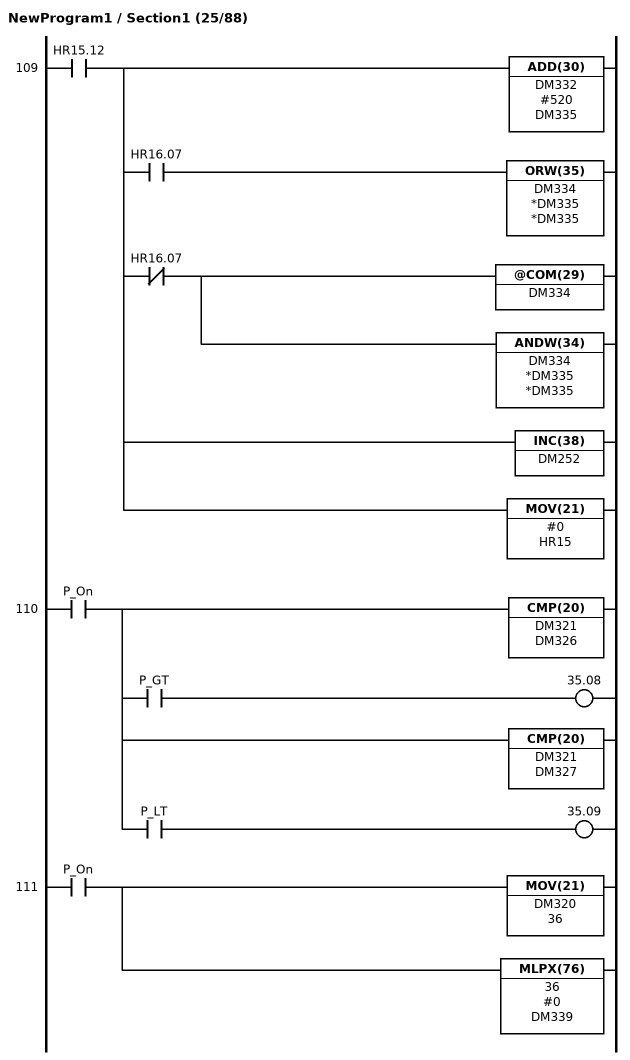
; [picture p24: NewProgram1 / Section1, rungs 109-111]
; rung 109
LD HR15.12
OUT TR0
ADD(30) DM332 #520 DM335
AND HR16.07
ORW(35) DM334 *DM335 *DM335
LD TR0
ANDNOT HR16.07
@COM(29) DM334
ANDW(34) DM334 *DM335 *DM335
LD TR0
INC(38) DM252
MOV(21) #0 HR15
; rung 110
LD P_On
OUT TR0
CMP(20) DM321 DM326
AND P_GT
OUT 35.08
LD TR0
CMP(20) DM321 DM327
AND P_LT
OUT 35.09
; rung 111
LD P_On
MOV(21) DM320 36
MLPX(76) 36 #0 DM339

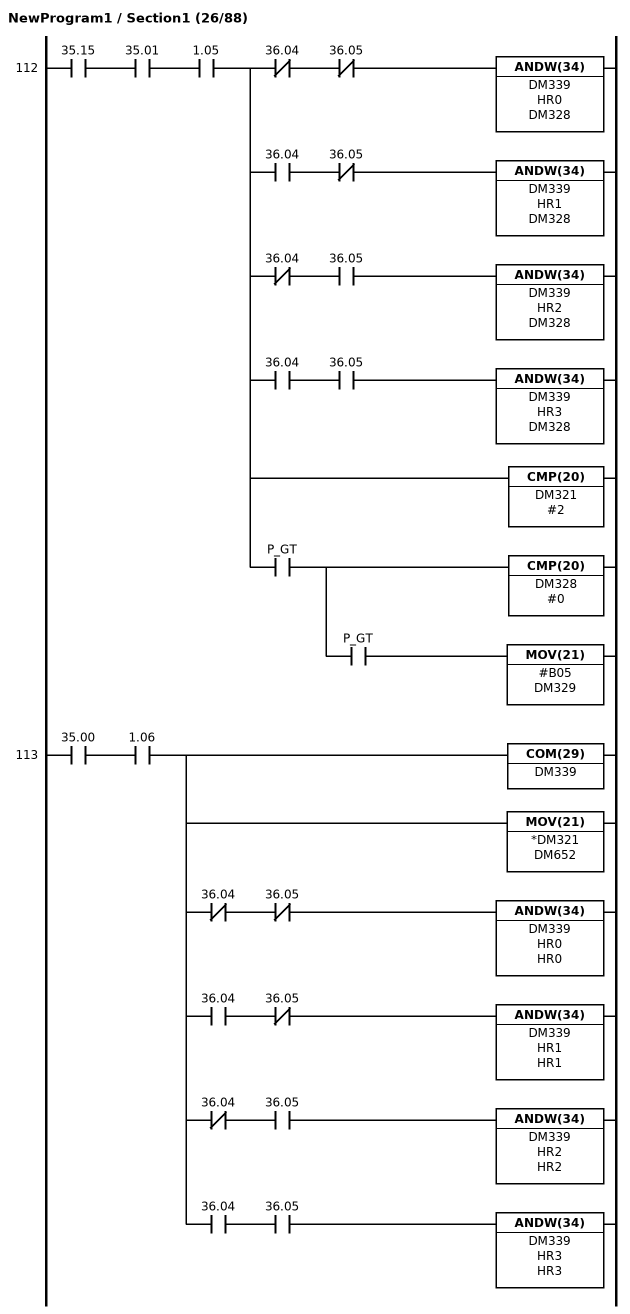
; rung 112
LD 35.15
AND 35.01
AND 1.05
OUT TR0
ANDNOT 36.04
ANDNOT 36.05
ANDW(34) DM339 HR0 DM328
LD TR0
AND 36.04
ANDNOT 36.05
ANDW(34) DM339 HR1 DM328
LD TR0
ANDNOT 36.04
AND 36.05
ANDW(34) DM339 HR2 DM328
LD TR0
AND 36.04
AND 36.05
ANDW(34) DM339 HR3 DM328
LD TR0
CMP(20) DM321 #2
AND P_GT
CMP(20) DM328 #0
AND P_GT
MOV(21) #B05 DM329
; rung 113
LD 35.00
AND 1.06
OUT TR0
COM(29) DM339
MOV(21) *DM321 DM652
ANDNOT 36.04
ANDNOT 36.05
ANDW(34) DM339 HR0 HR0
LD TR0
AND 36.04
ANDNOT 36.05
ANDW(34) DM339 HR1 HR1
LD TR0
ANDNOT 36.04
AND 36.05
ANDW(34) DM339 HR2 HR2
LD TR0
AND 36.04
AND 36.05
ANDW(34) DM339 HR3 HR3

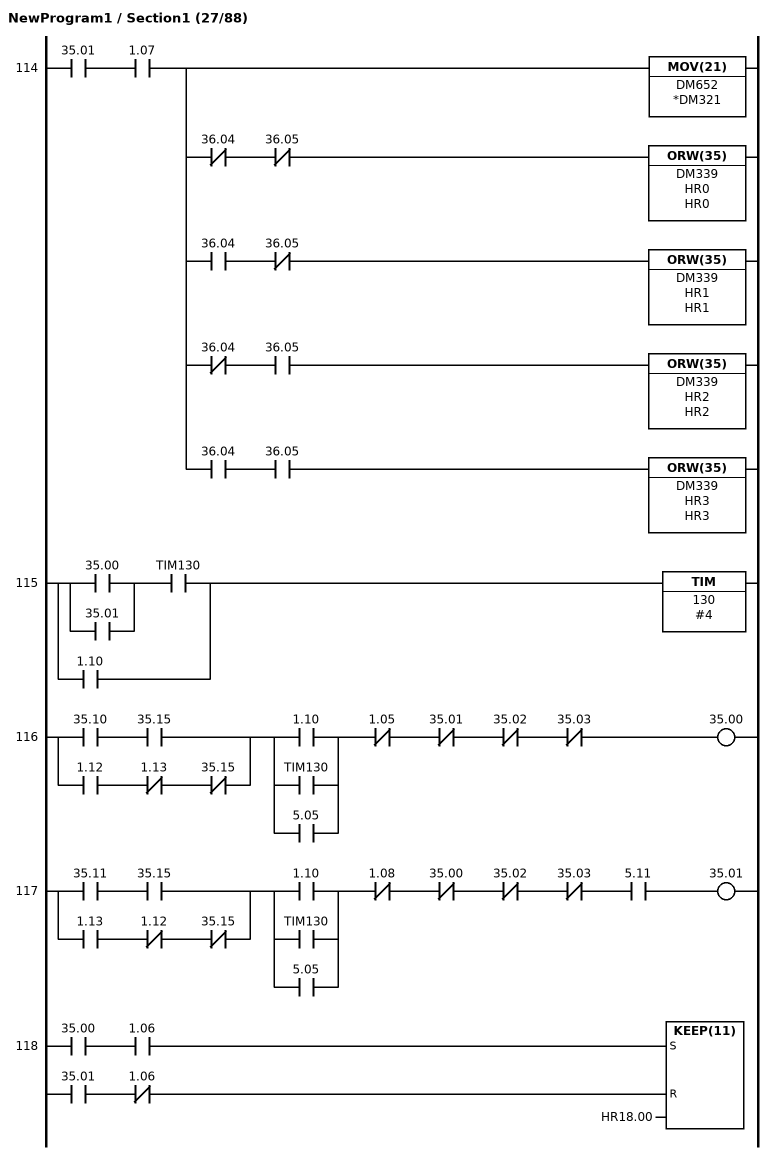
; rung 114
LD 35.01
AND 1.07
OUT TR0
MOV(21) DM652 *DM321
ANDNOT 36.04
ANDNOT 36.05
ORW(35) DM339 HR0 HR0
LD TR0
AND 36.04
ANDNOT 36.05
ORW(35) DM339 HR1 HR1
LD TR0
ANDNOT 36.04
AND 36.05
ORW(35) DM339 HR2 HR2
LD TR0
AND 36.04
AND 36.05
ORW(35) DM339 HR3 HR3
; rung 115
LD 35.00
OR 35.01
AND TIM130
OR 1.10
TIM 130 #4
; rung 116
LD 35.10
AND 35.15
LD 1.12
ANDNOT 1.13
ANDNOT 35.15
ORLD
LD 1.10
OR TIM130
OR 5.05
ANDLD
ANDNOT 1.05
ANDNOT 35.01
ANDNOT 35.02
ANDNOT 35.03
OUT 35.00
; rung 117
LD 35.11
AND 35.15
LD 1.13
ANDNOT 1.12
ANDNOT 35.15
ORLD
LD 1.10
OR TIM130
OR 5.05
ANDLD
ANDNOT 1.08
ANDNOT 35.00
ANDNOT 35.02
ANDNOT 35.03
AND 5.11
OUT 35.01
; rung 118
LD 35.00
AND 1.06
LD 35.01
ANDNOT 1.06
KEEP(11) HR18.00

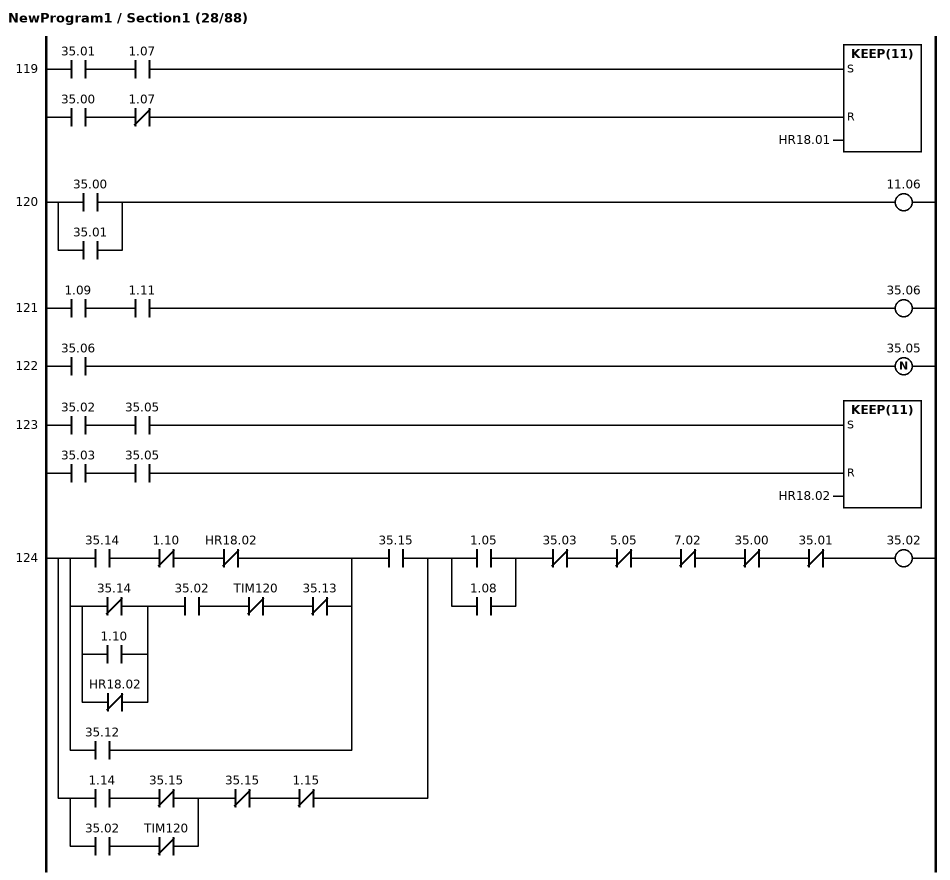
; rung 119
LD 35.01
AND 1.07
LD 35.00
ANDNOT 1.07
KEEP(11) HR18.01
; rung 120
LD 35.00
OR 35.01
OUT 11.06
; rung 121
LD 1.09
AND 1.11
OUT 35.06
; rung 122
LD 35.06
DIFD(14) 35.05
; rung 123
LD 35.02
AND 35.05
LD 35.03
AND 35.05
KEEP(11) HR18.02
; rung 124
LD 35.14
ANDNOT 1.10
ANDNOT HR18.02
LDNOT 35.14
OR 1.10
ORNOT HR18.02
AND 35.02
ANDNOT TIM120
ANDNOT 35.13
ORLD
OR 35.12
AND 35.15
LD 1.14
ANDNOT 35.15
LD 35.02
ANDNOT TIM120
ORLD
ANDNOT 35.15
ANDNOT 1.15
ORLD
LD 1.05
OR 1.08
ANDLD
ANDNOT 35.03
ANDNOT 5.05
ANDNOT 7.02
ANDNOT 35.00
ANDNOT 35.01
OUT 35.02

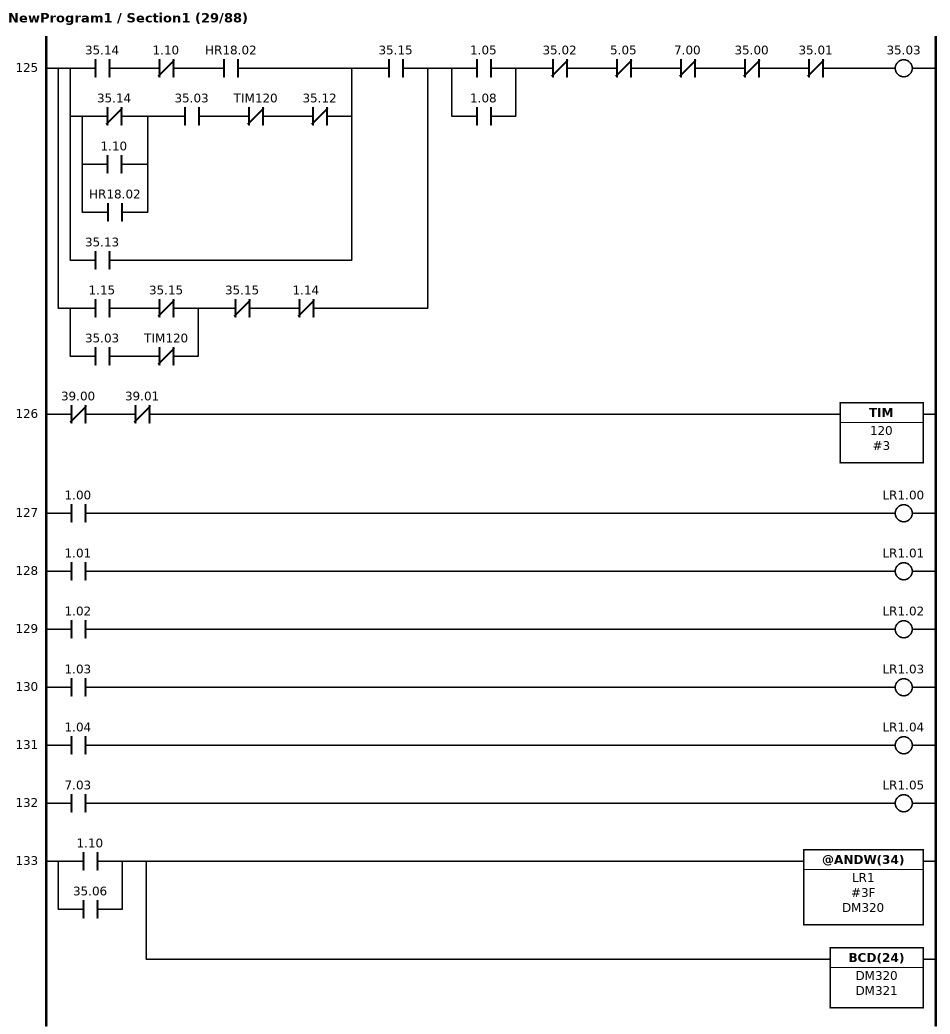
; rung 125
LD 35.14
ANDNOT 1.10
AND HR18.02
LDNOT 35.14
OR 1.10
OR HR18.02
AND 35.03
ANDNOT TIM120
ANDNOT 35.12
ORLD
OR 35.13
AND 35.15
LD 1.15
ANDNOT 35.15
LD 35.03
ANDNOT TIM120
ORLD
ANDNOT 35.15
ANDNOT 1.14
ORLD
LD 1.05
OR 1.08
ANDLD
ANDNOT 35.02
ANDNOT 5.05
ANDNOT 7.00
ANDNOT 35.00
ANDNOT 35.01
OUT 35.03
; rung 126
LDNOT 39.00
ANDNOT 39.01
TIM 120 #3
; rung 127
LD 1.00
OUT LR1.00
; rung 128
LD 1.01
OUT LR1.01
; rung 129
LD 1.02
OUT LR1.02
; rung 130
LD 1.03
OUT LR1.03
; rung 131
LD 1.04
OUT LR1.04
; rung 132
LD 7.03
OUT LR1.05
; rung 133
LD 1.10
OR 35.06
@ANDW(34) LR1 #3F DM320
BCD(24) DM320 DM321

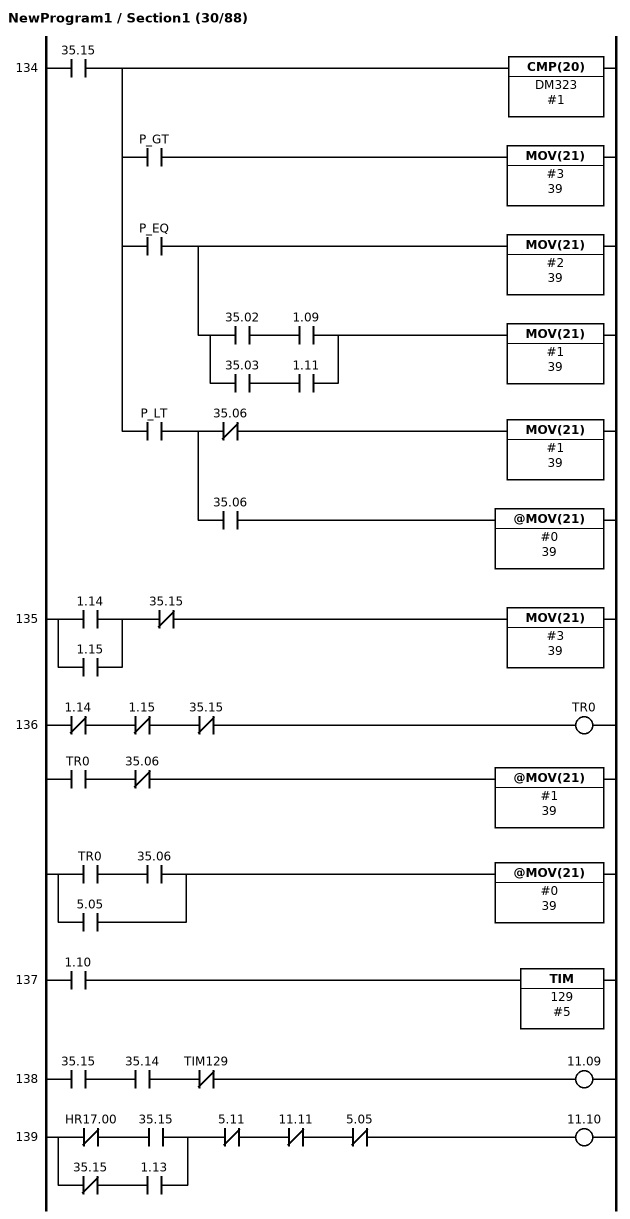
; rung 134
LD 35.15
OUT TR0
CMP(20) DM323 #1
AND P_GT
MOV(21) #3 39
LD TR0
AND P_EQ
MOV(21) #2 39
LD 35.02
AND 1.09
LD 35.03
AND 1.11
ORLD
ANDLD
MOV(21) #1 39
LD TR0
AND P_LT
OUT TR0
ANDNOT 35.06
MOV(21) #1 39
LD TR0
AND 35.06
@MOV(21) #0 39
; rung 135
LD 1.14
OR 1.15
ANDNOT 35.15
MOV(21) #3 39
; rung 136
LDNOT 1.14
ANDNOT 1.15
ANDNOT 35.15
OUT TR0
ANDNOT 35.06
@MOV(21) #1 39
LD TR0
AND 35.06
OR 5.05
@MOV(21) #0 39
; rung 137
LD 1.10
TIM 129 #5
; rung 138
LD 35.15
AND 35.14
ANDNOT TIM129
OUT 11.09
; rung 139
LDNOT HR17.00
AND 35.15
LDNOT 35.15
AND 1.13
ORLD
ANDNOT 5.11
ANDNOT 11.11
ANDNOT 5.05
OUT 11.10

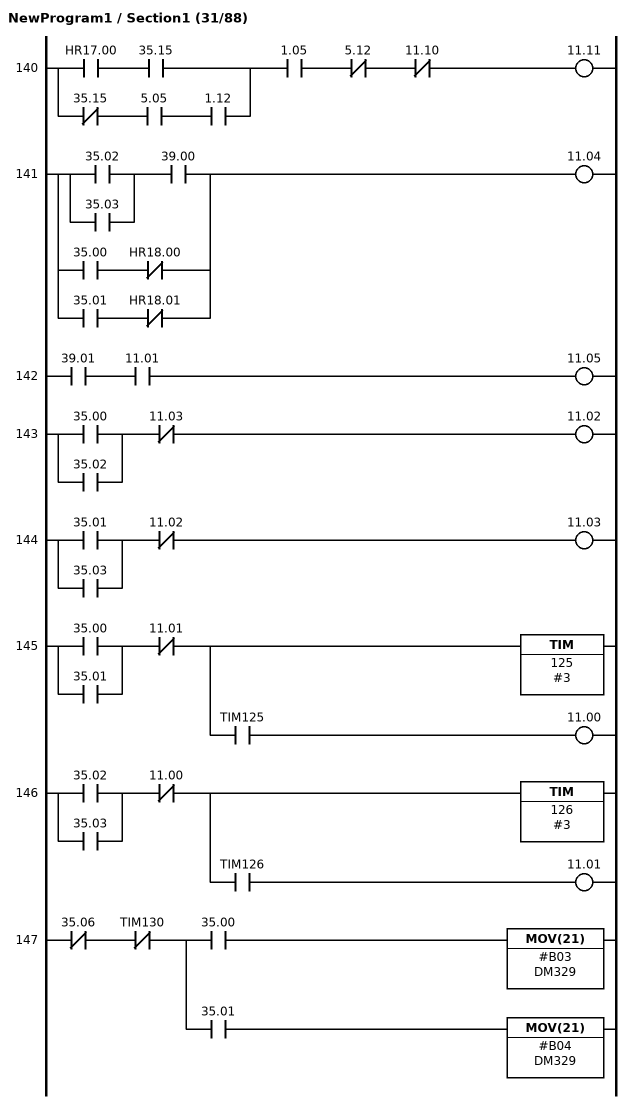
; rung 140
LD HR17.00
AND 35.15
LDNOT 35.15
AND 5.05
AND 1.12
ORLD
AND 1.05
ANDNOT 5.12
ANDNOT 11.10
OUT 11.11
; rung 141
LD 35.02
OR 35.03
AND 39.00
LD 35.00
ANDNOT HR18.00
ORLD
LD 35.01
ANDNOT HR18.01
ORLD
OUT 11.04
; rung 142
LD 39.01
AND 11.01
OUT 11.05
; rung 143
LD 35.00
OR 35.02
ANDNOT 11.03
OUT 11.02
; rung 144
LD 35.01
OR 35.03
ANDNOT 11.02
OUT 11.03
; rung 145
LD 35.00
OR 35.01
ANDNOT 11.01
TIM 125 #3
AND TIM125
OUT 11.00
; rung 146
LD 35.02
OR 35.03
ANDNOT 11.00
TIM 126 #3
AND TIM126
OUT 11.01
; rung 147
LDNOT 35.06
ANDNOT TIM130
OUT TR0
AND 35.00
MOV(21) #B03 DM329
LD TR0
AND 35.01
MOV(21) #B04 DM329

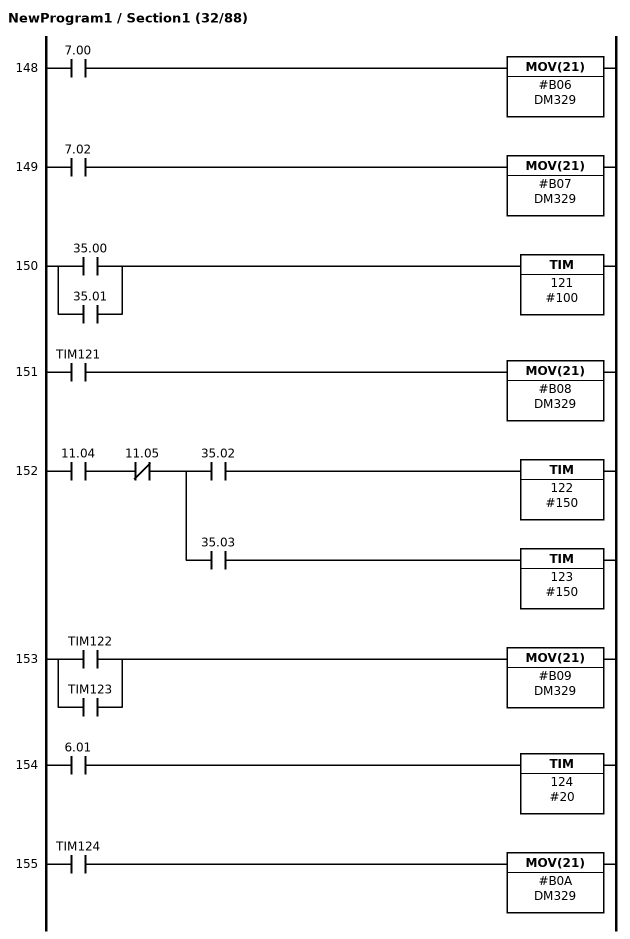
; rung 148
LD 7.00
MOV(21) #B06 DM329
; rung 149
LD 7.02
MOV(21) #B07 DM329
; rung 150
LD 35.00
OR 35.01
TIM 121 #100
; rung 151
LD TIM121
MOV(21) #B08 DM329
; rung 152
LD 11.04
ANDNOT 11.05
OUT TR0
AND 35.02
TIM 122 #150
LD TR0
AND 35.03
TIM 123 #150
; rung 153
LD TIM122
OR TIM123
MOV(21) #B09 DM329
; rung 154
LD 6.01
TIM 124 #20
; rung 155
LD TIM124
MOV(21) #B0A DM329

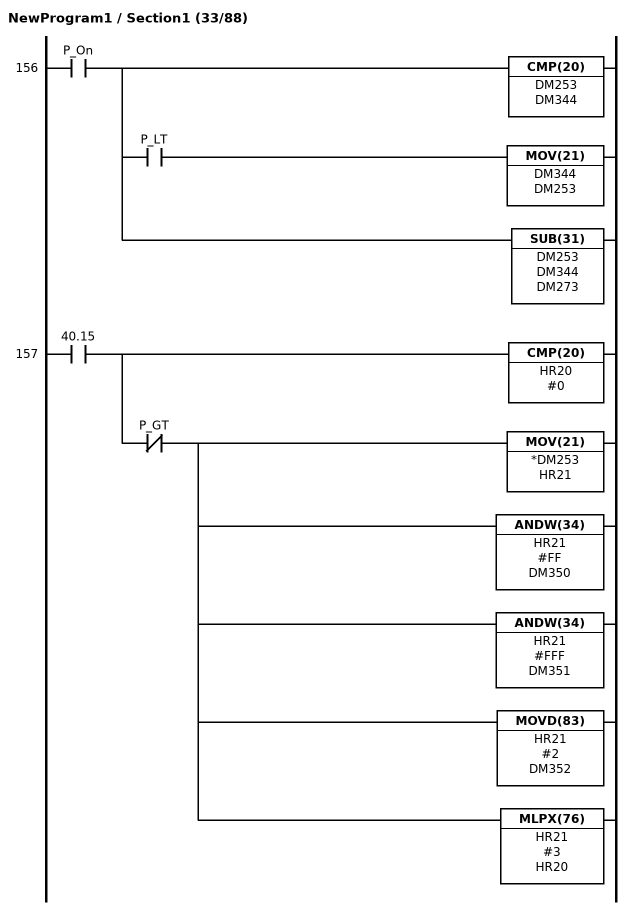
; rung 156
LD P_On
OUT TR0
CMP(20) DM253 DM344
AND P_LT
MOV(21) DM344 DM253
LD TR0
SUB(31) DM253 DM344 DM273
; rung 157
LD 40.15
CMP(20) HR20 #0
ANDNOT P_GT
MOV(21) *DM253 HR21
ANDW(34) HR21 #FF DM350
ANDW(34) HR21 #FFF DM351
MOVD(83) HR21 #2 DM352
MLPX(76) HR21 #3 HR20

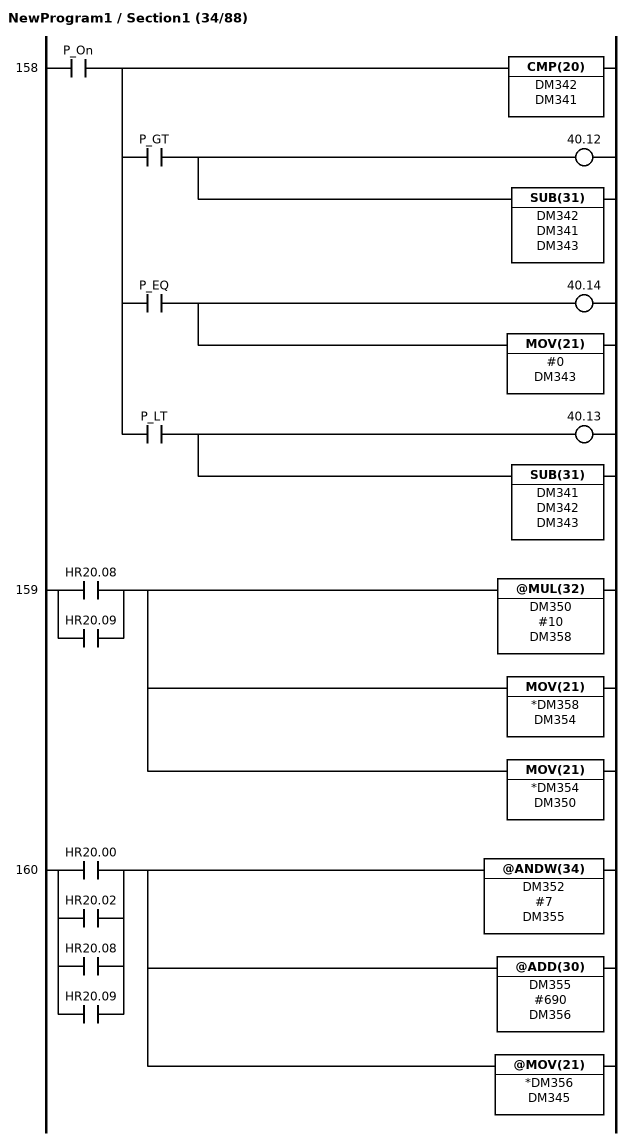
; rung 158
LD P_On
OUT TR0
CMP(20) DM342 DM341
AND P_GT
OUT 40.12
SUB(31) DM342 DM341 DM343
LD TR0
AND P_EQ
OUT 40.14
MOV(21) #0 DM343
LD TR0
AND P_LT
OUT 40.13
SUB(31) DM341 DM342 DM343
; rung 159
LD HR20.08
OR HR20.09
@MUL(32) DM350 #10 DM358
MOV(21) *DM358 DM354
MOV(21) *DM354 DM350
; rung 160
LD HR20.00
OR HR20.02
OR HR20.08
OR HR20.09
@ANDW(34) DM352 #7 DM355
@ADD(30) DM355 #690 DM356
@MOV(21) *DM356 DM345

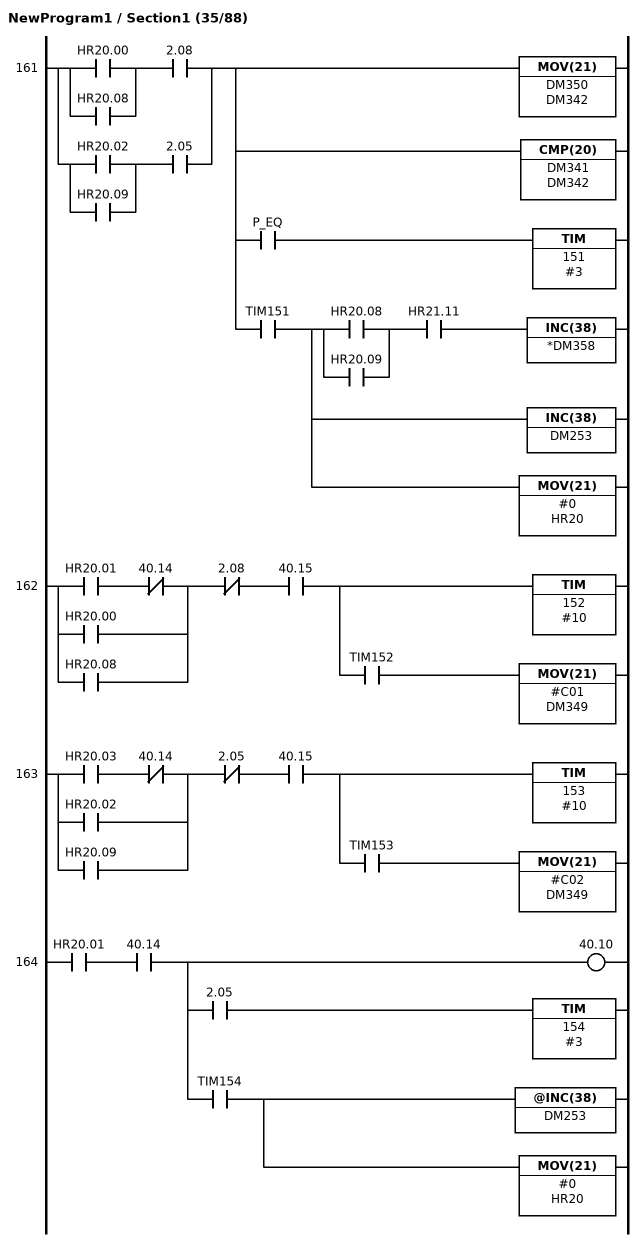
; rung 161
LD HR20.00
OR HR20.08
AND 2.08
LD HR20.02
OR HR20.09
AND 2.05
ORLD
OUT TR0
MOV(21) DM350 DM342
CMP(20) DM341 DM342
AND P_EQ
TIM 151 #3
LD TR0
AND TIM151
OUT TR0
LD HR20.08
OR HR20.09
ANDLD
AND HR21.11
INC(38) *DM358
LD TR0
INC(38) DM253
MOV(21) #0 HR20
; rung 162
LD HR20.01
ANDNOT 40.14
OR HR20.00
OR HR20.08
ANDNOT 2.08
AND 40.15
TIM 152 #10
AND TIM152
MOV(21) #C01 DM349
; rung 163
LD HR20.03
ANDNOT 40.14
OR HR20.02
OR HR20.09
ANDNOT 2.05
AND 40.15
TIM 153 #10
AND TIM153
MOV(21) #C02 DM349
; rung 164
LD HR20.01
AND 40.14
OUT TR0
OUT 40.10
AND 2.05
TIM 154 #3
LD TR0
AND TIM154
@INC(38) DM253
MOV(21) #0 HR20

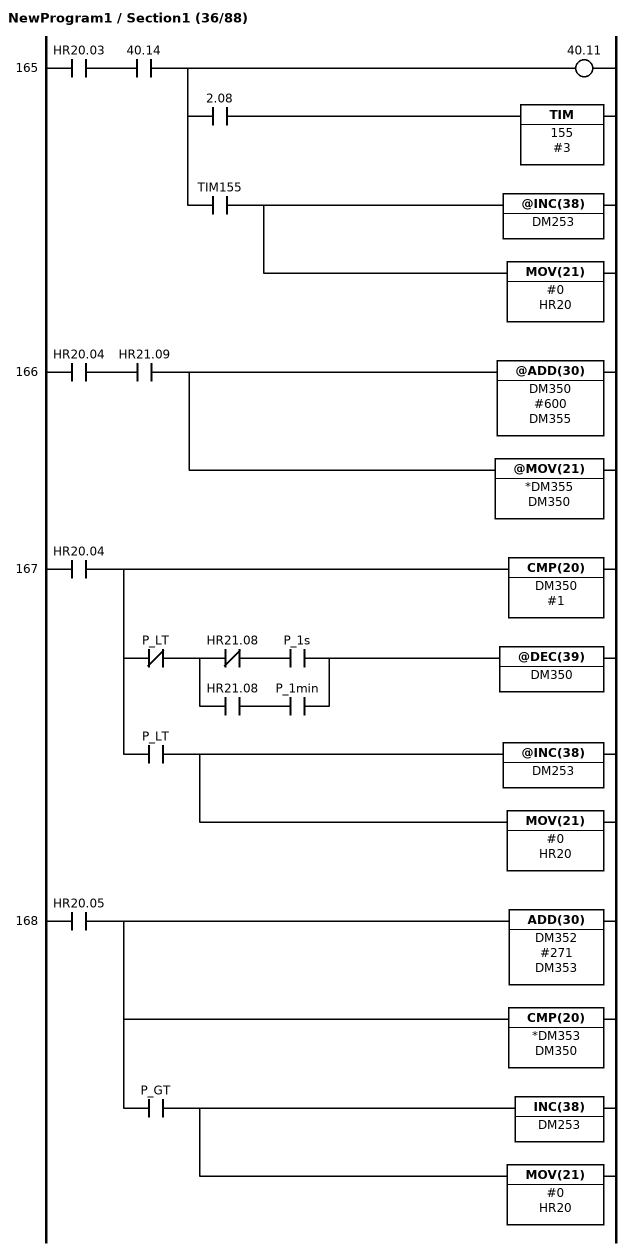
; rung 165
LD HR20.03
AND 40.14
OUT TR0
OUT 40.11
AND 2.08
TIM 155 #3
LD TR0
AND TIM155
@INC(38) DM253
MOV(21) #0 HR20
; rung 166
LD HR20.04
AND HR21.09
@ADD(30) DM350 #600 DM355
@MOV(21) *DM355 DM350
; rung 167
LD HR20.04
OUT TR0
CMP(20) DM350 #1
ANDNOT P_LT
LDNOT HR21.08
AND P_1s
LD HR21.08
AND P_1min
ORLD
ANDLD
@DEC(39) DM350
LD TR0
AND P_LT
@INC(38) DM253
MOV(21) #0 HR20
; rung 168
LD HR20.05
ADD(30) DM352 #271 DM353
CMP(20) *DM353 DM350
AND P_GT
INC(38) DM253
MOV(21) #0 HR20

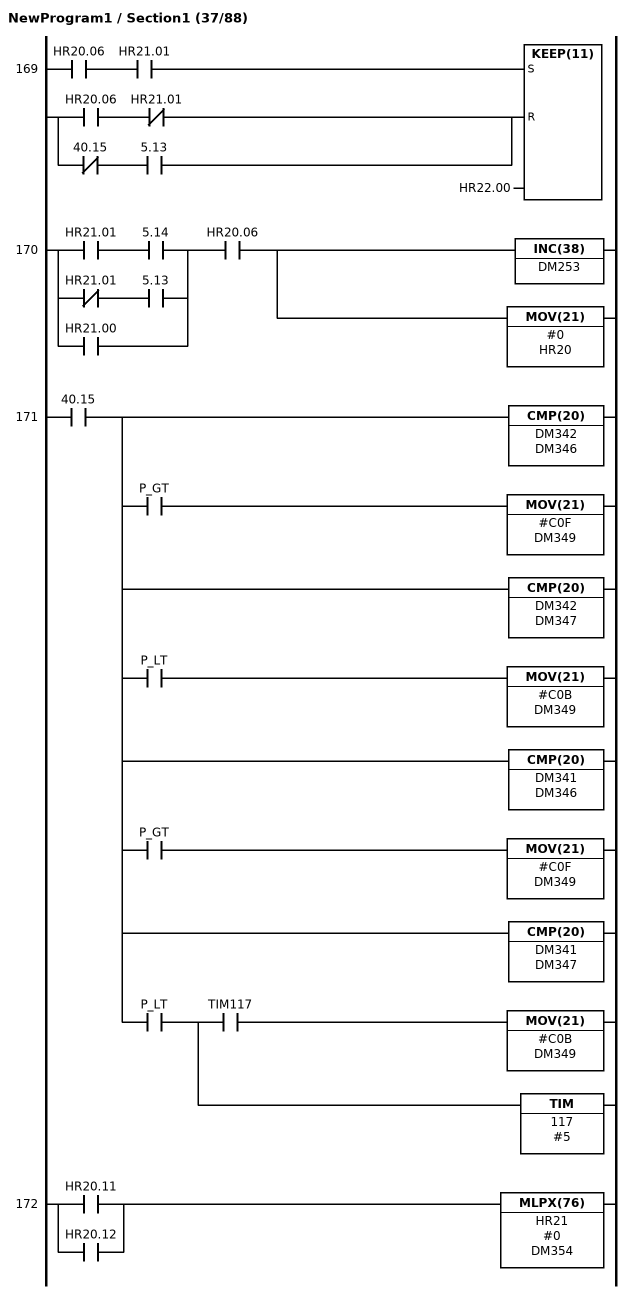
; rung 169
LD HR20.06
AND HR21.01
LD HR20.06
ANDNOT HR21.01
LDNOT 40.15
AND 5.13
ORLD
KEEP(11) HR22.00
; rung 170
LD HR21.01
AND 5.14
LDNOT HR21.01
AND 5.13
ORLD
OR HR21.00
AND HR20.06
INC(38) DM253
MOV(21) #0 HR20
; rung 171
LD 40.15
OUT TR0
CMP(20) DM342 DM346
AND P_GT
MOV(21) #C0F DM349
LD TR0
CMP(20) DM342 DM347
AND P_LT
MOV(21) #C0B DM349
LD TR0
CMP(20) DM341 DM346
AND P_GT
MOV(21) #C0F DM349
LD TR0
CMP(20) DM341 DM347
AND P_LT
OUT TR0
AND TIM117
MOV(21) #C0B DM349
LD TR0
TIM 117 #5
; rung 172
LD HR20.11
OR HR20.12
MLPX(76) HR21 #0 DM354

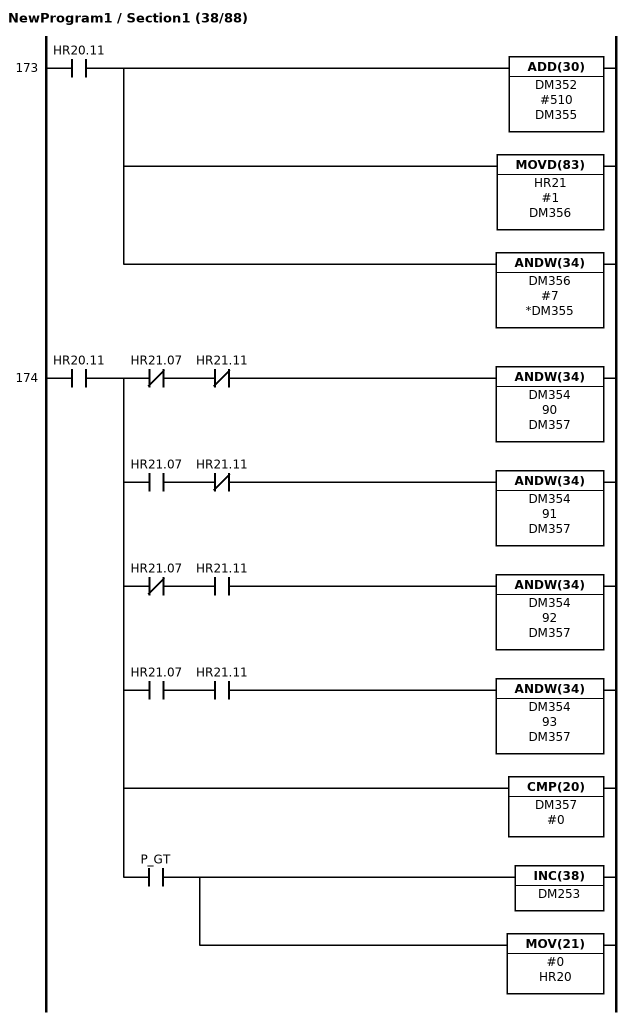
; rung 173
LD HR20.11
ADD(30) DM352 #510 DM355
MOVD(83) HR21 #1 DM356
ANDW(34) DM356 #7 *DM355
; rung 174
LD HR20.11
OUT TR0
ANDNOT HR21.07
ANDNOT HR21.11
ANDW(34) DM354 90 DM357
LD TR0
AND HR21.07
ANDNOT HR21.11
ANDW(34) DM354 91 DM357
LD TR0
ANDNOT HR21.07
AND HR21.11
ANDW(34) DM354 92 DM357
LD TR0
AND HR21.07
AND HR21.11
ANDW(34) DM354 93 DM357
LD TR0
CMP(20) DM357 #0
AND P_GT
INC(38) DM253
MOV(21) #0 HR20

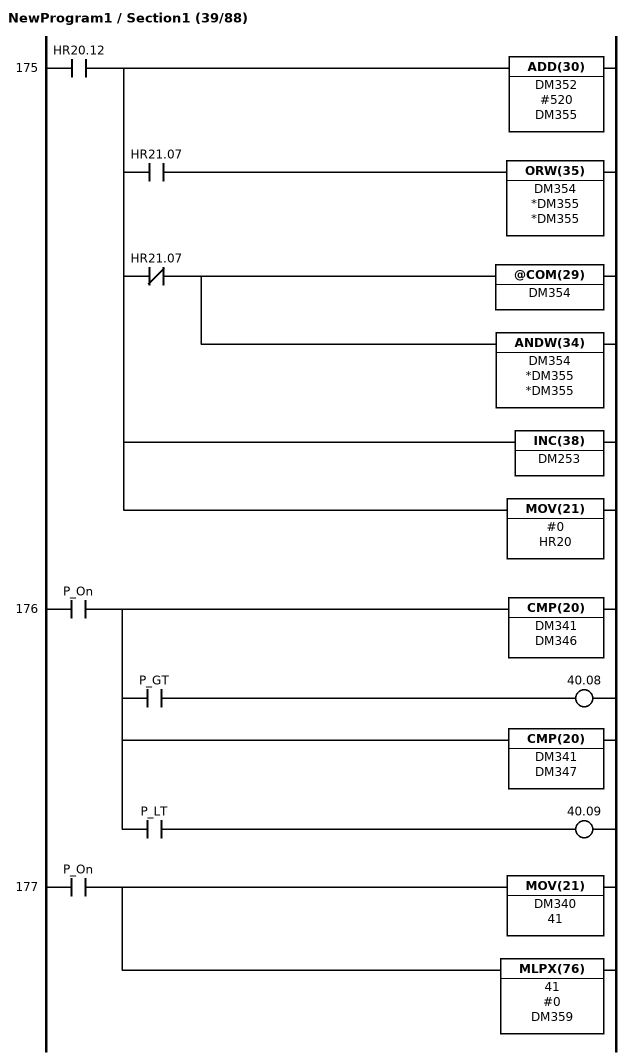
; rung 175
LD HR20.12
OUT TR0
ADD(30) DM352 #520 DM355
AND HR21.07
ORW(35) DM354 *DM355 *DM355
LD TR0
ANDNOT HR21.07
@COM(29) DM354
ANDW(34) DM354 *DM355 *DM355
LD TR0
INC(38) DM253
MOV(21) #0 HR20
; rung 176
LD P_On
OUT TR0
CMP(20) DM341 DM346
AND P_GT
OUT 40.08
LD TR0
CMP(20) DM341 DM347
AND P_LT
OUT 40.09
; rung 177
LD P_On
MOV(21) DM340 41
MLPX(76) 41 #0 DM359

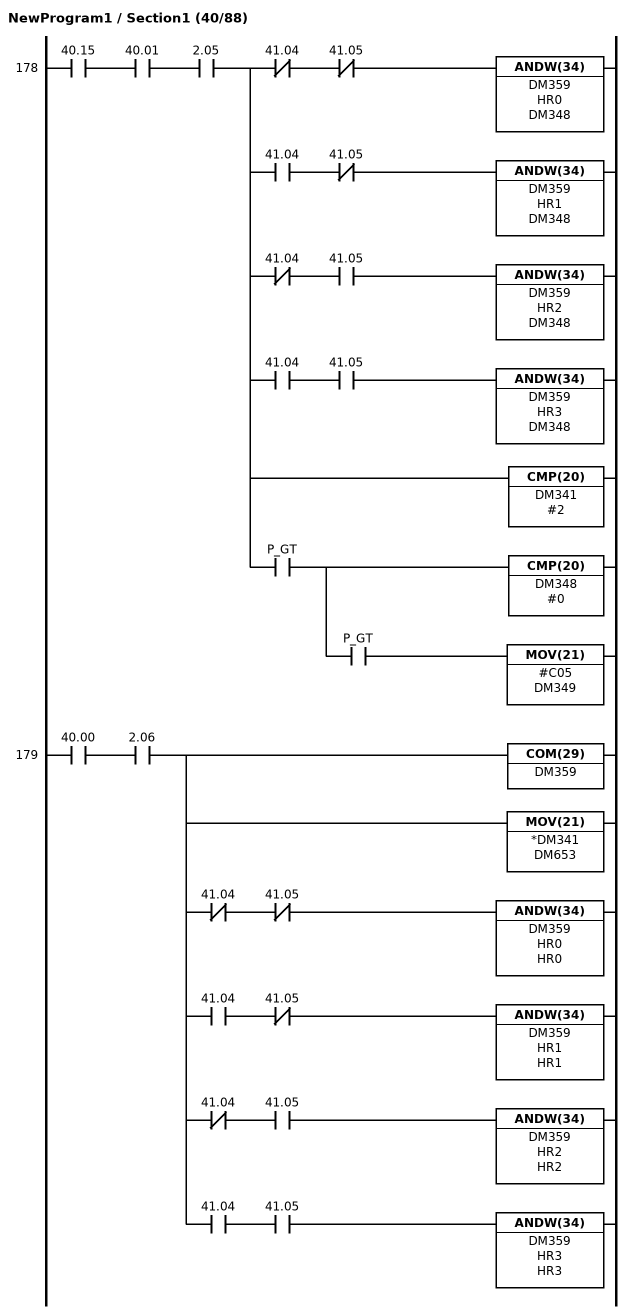
; rung 178
LD 40.15
AND 40.01
AND 2.05
OUT TR0
ANDNOT 41.04
ANDNOT 41.05
ANDW(34) DM359 HR0 DM348
LD TR0
AND 41.04
ANDNOT 41.05
ANDW(34) DM359 HR1 DM348
LD TR0
ANDNOT 41.04
AND 41.05
ANDW(34) DM359 HR2 DM348
LD TR0
AND 41.04
AND 41.05
ANDW(34) DM359 HR3 DM348
LD TR0
CMP(20) DM341 #2
AND P_GT
CMP(20) DM348 #0
AND P_GT
MOV(21) #C05 DM349
; rung 179
LD 40.00
AND 2.06
OUT TR0
COM(29) DM359
MOV(21) *DM341 DM653
ANDNOT 41.04
ANDNOT 41.05
ANDW(34) DM359 HR0 HR0
LD TR0
AND 41.04
ANDNOT 41.05
ANDW(34) DM359 HR1 HR1
LD TR0
ANDNOT 41.04
AND 41.05
ANDW(34) DM359 HR2 HR2
LD TR0
AND 41.04
AND 41.05
ANDW(34) DM359 HR3 HR3

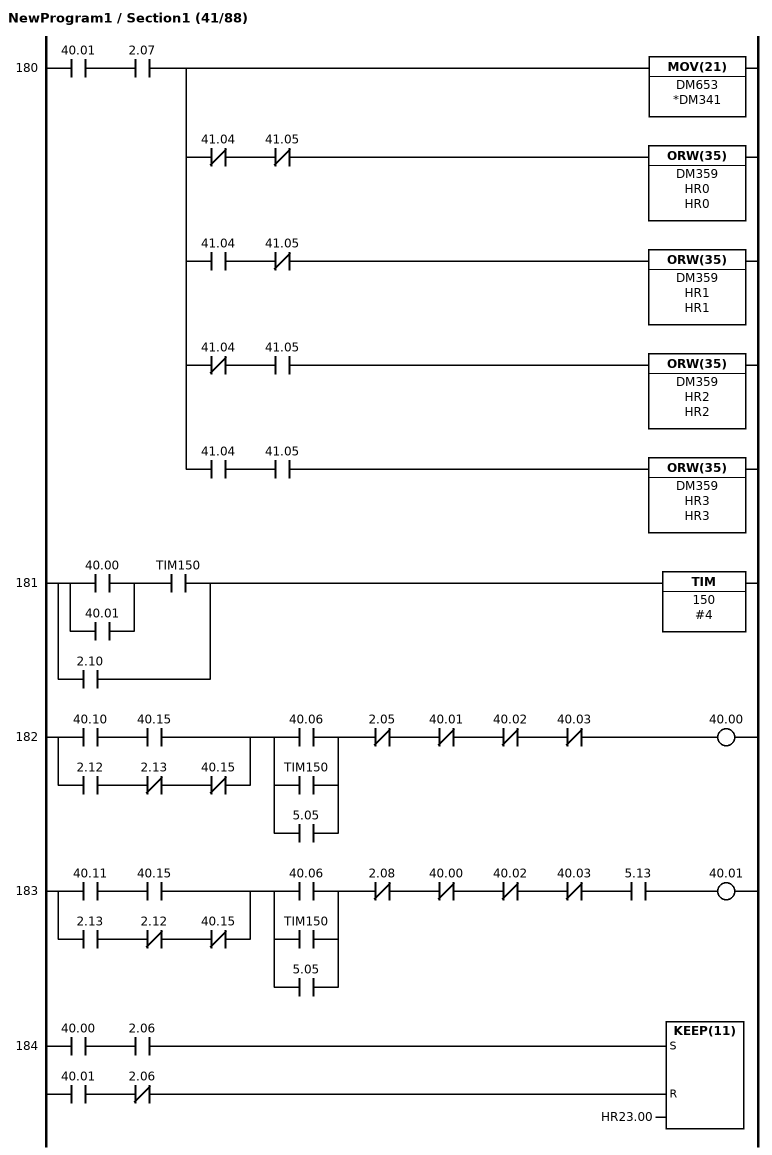
; rung 180
LD 40.01
AND 2.07
OUT TR0
MOV(21) DM653 *DM341
ANDNOT 41.04
ANDNOT 41.05
ORW(35) DM359 HR0 HR0
LD TR0
AND 41.04
ANDNOT 41.05
ORW(35) DM359 HR1 HR1
LD TR0
ANDNOT 41.04
AND 41.05
ORW(35) DM359 HR2 HR2
LD TR0
AND 41.04
AND 41.05
ORW(35) DM359 HR3 HR3
; rung 181
LD 40.00
OR 40.01
AND TIM150
OR 2.10
TIM 150 #4
; rung 182
LD 40.10
AND 40.15
LD 2.12
ANDNOT 2.13
ANDNOT 40.15
ORLD
LD 40.06
OR TIM150
OR 5.05
ANDLD
ANDNOT 2.05
ANDNOT 40.01
ANDNOT 40.02
ANDNOT 40.03
OUT 40.00
; rung 183
LD 40.11
AND 40.15
LD 2.13
ANDNOT 2.12
ANDNOT 40.15
ORLD
LD 40.06
OR TIM150
OR 5.05
ANDLD
ANDNOT 2.08
ANDNOT 40.00
ANDNOT 40.02
ANDNOT 40.03
AND 5.13
OUT 40.01
; rung 184
LD 40.00
AND 2.06
LD 40.01
ANDNOT 2.06
KEEP(11) HR23.00

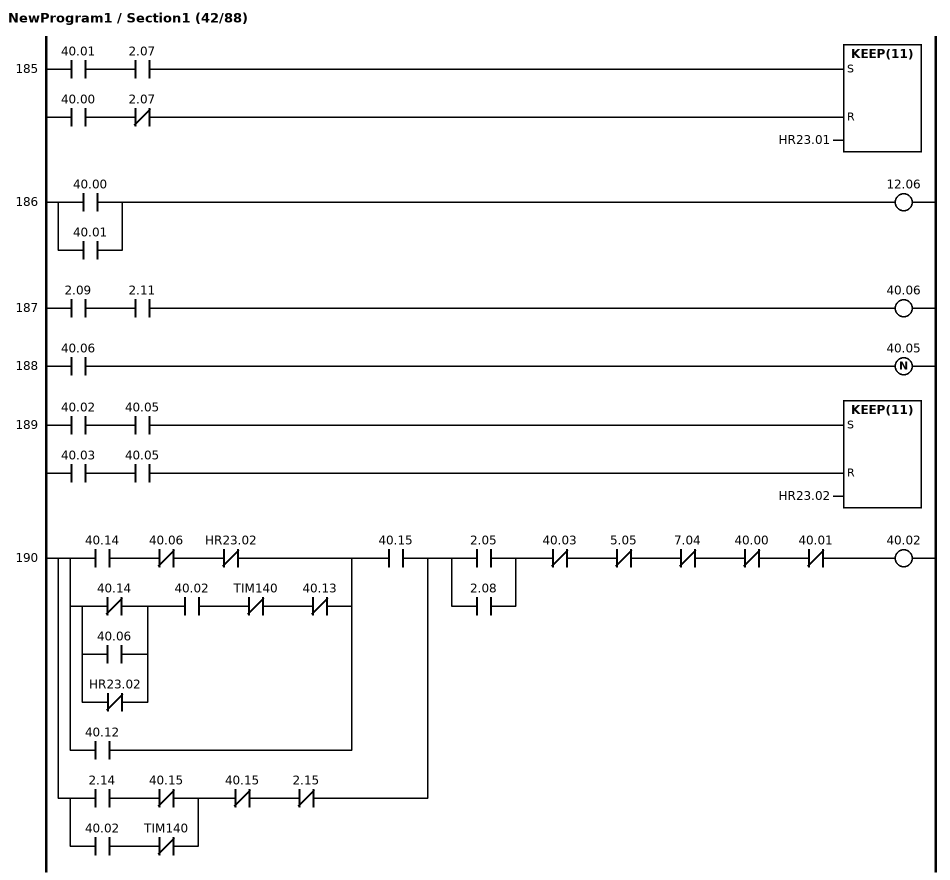
; rung 185
LD 40.01
AND 2.07
LD 40.00
ANDNOT 2.07
KEEP(11) HR23.01
; rung 186
LD 40.00
OR 40.01
OUT 12.06
; rung 187
LD 2.09
AND 2.11
OUT 40.06
; rung 188
LD 40.06
DIFD(14) 40.05
; rung 189
LD 40.02
AND 40.05
LD 40.03
AND 40.05
KEEP(11) HR23.02
; rung 190
LD 40.14
ANDNOT 40.06
ANDNOT HR23.02
LDNOT 40.14
OR 40.06
ORNOT HR23.02
AND 40.02
ANDNOT TIM140
ANDNOT 40.13
ORLD
OR 40.12
AND 40.15
LD 2.14
ANDNOT 40.15
LD 40.02
ANDNOT TIM140
ORLD
ANDNOT 40.15
ANDNOT 2.15
ORLD
LD 2.05
OR 2.08
ANDLD
ANDNOT 40.03
ANDNOT 5.05
ANDNOT 7.04
ANDNOT 40.00
ANDNOT 40.01
OUT 40.02

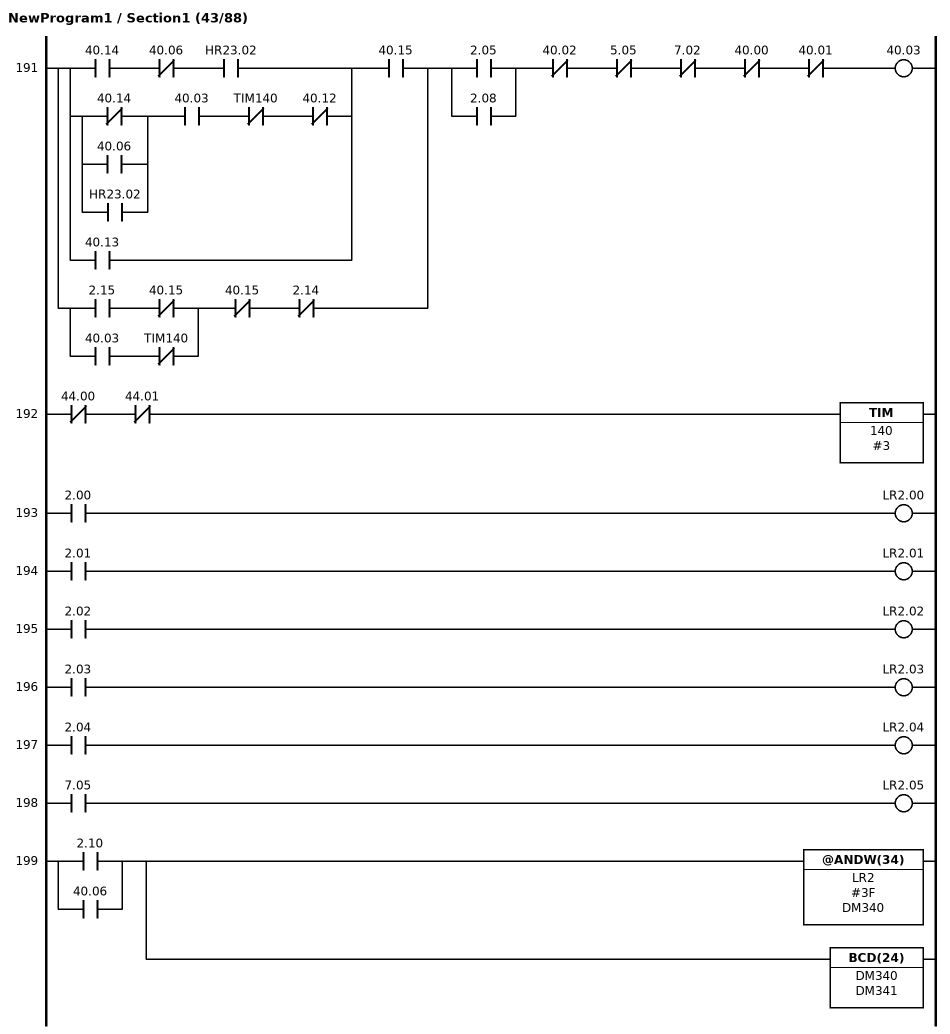
; rung 191
LD 40.14
ANDNOT 40.06
AND HR23.02
LDNOT 40.14
OR 40.06
OR HR23.02
AND 40.03
ANDNOT TIM140
ANDNOT 40.12
ORLD
OR 40.13
AND 40.15
LD 2.15
ANDNOT 40.15
LD 40.03
ANDNOT TIM140
ORLD
ANDNOT 40.15
ANDNOT 2.14
ORLD
LD 2.05
OR 2.08
ANDLD
ANDNOT 40.02
ANDNOT 5.05
ANDNOT 7.02
ANDNOT 40.00
ANDNOT 40.01
OUT 40.03
; rung 192
LDNOT 44.00
ANDNOT 44.01
TIM 140 #3
; rung 193
LD 2.00
OUT LR2.00
; rung 194
LD 2.01
OUT LR2.01
; rung 195
LD 2.02
OUT LR2.02
; rung 196
LD 2.03
OUT LR2.03
; rung 197
LD 2.04
OUT LR2.04
; rung 198
LD 7.05
OUT LR2.05
; rung 199
LD 2.10
OR 40.06
@ANDW(34) LR2 #3F DM340
BCD(24) DM340 DM341

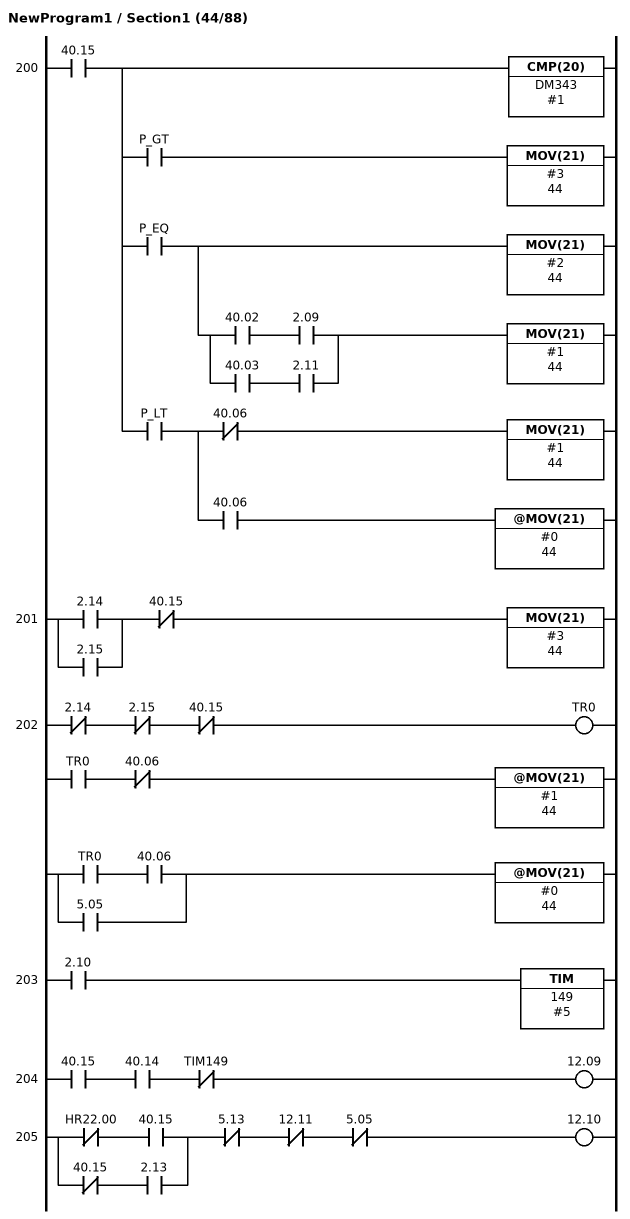
; rung 200
LD 40.15
OUT TR0
CMP(20) DM343 #1
AND P_GT
MOV(21) #3 44
LD TR0
AND P_EQ
MOV(21) #2 44
LD 40.02
AND 2.09
LD 40.03
AND 2.11
ORLD
ANDLD
MOV(21) #1 44
LD TR0
AND P_LT
OUT TR0
ANDNOT 40.06
MOV(21) #1 44
LD TR0
AND 40.06
@MOV(21) #0 44
; rung 201
LD 2.14
OR 2.15
ANDNOT 40.15
MOV(21) #3 44
; rung 202
LDNOT 2.14
ANDNOT 2.15
ANDNOT 40.15
OUT TR0
ANDNOT 40.06
@MOV(21) #1 44
LD TR0
AND 40.06
OR 5.05
@MOV(21) #0 44
; rung 203
LD 2.10
TIM 149 #5
; rung 204
LD 40.15
AND 40.14
ANDNOT TIM149
OUT 12.09
; rung 205
LDNOT HR22.00
AND 40.15
LDNOT 40.15
AND 2.13
ORLD
ANDNOT 5.13
ANDNOT 12.11
ANDNOT 5.05
OUT 12.10

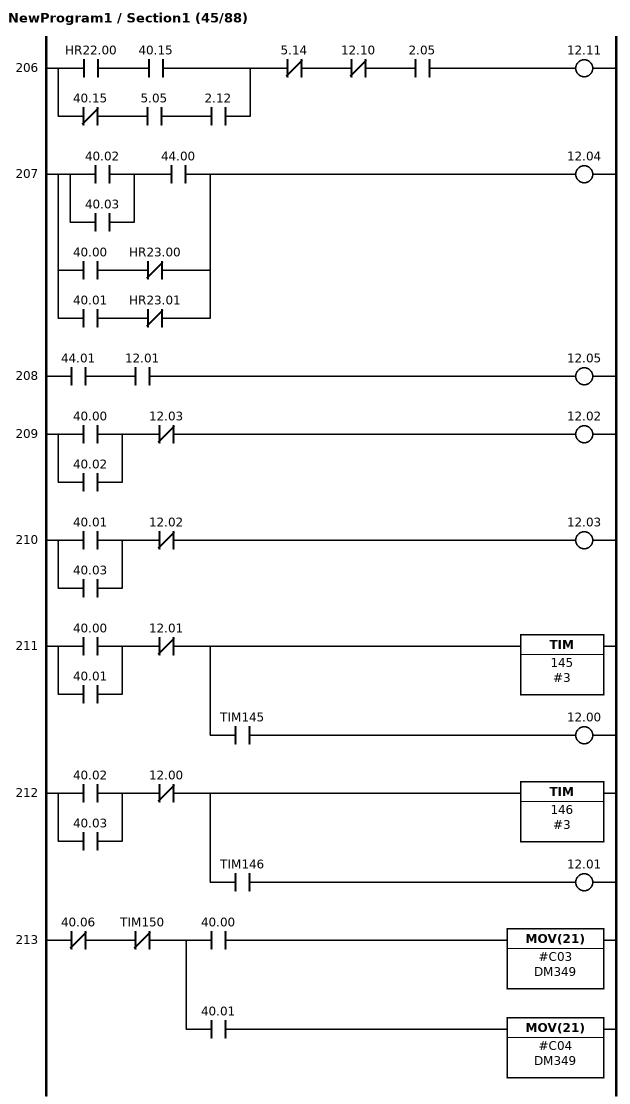
; rung 206
LD HR22.00
AND 40.15
LDNOT 40.15
AND 5.05
AND 2.12
ORLD
ANDNOT 5.14
ANDNOT 12.10
AND 2.05
OUT 12.11
; rung 207
LD 40.02
OR 40.03
AND 44.00
LD 40.00
ANDNOT HR23.00
ORLD
LD 40.01
ANDNOT HR23.01
ORLD
OUT 12.04
; rung 208
LD 44.01
AND 12.01
OUT 12.05
; rung 209
LD 40.00
OR 40.02
ANDNOT 12.03
OUT 12.02
; rung 210
LD 40.01
OR 40.03
ANDNOT 12.02
OUT 12.03
; rung 211
LD 40.00
OR 40.01
ANDNOT 12.01
TIM 145 #3
AND TIM145
OUT 12.00
; rung 212
LD 40.02
OR 40.03
ANDNOT 12.00
TIM 146 #3
AND TIM146
OUT 12.01
; rung 213
LDNOT 40.06
ANDNOT TIM150
OUT TR0
AND 40.00
MOV(21) #C03 DM349
LD TR0
AND 40.01
MOV(21) #C04 DM349

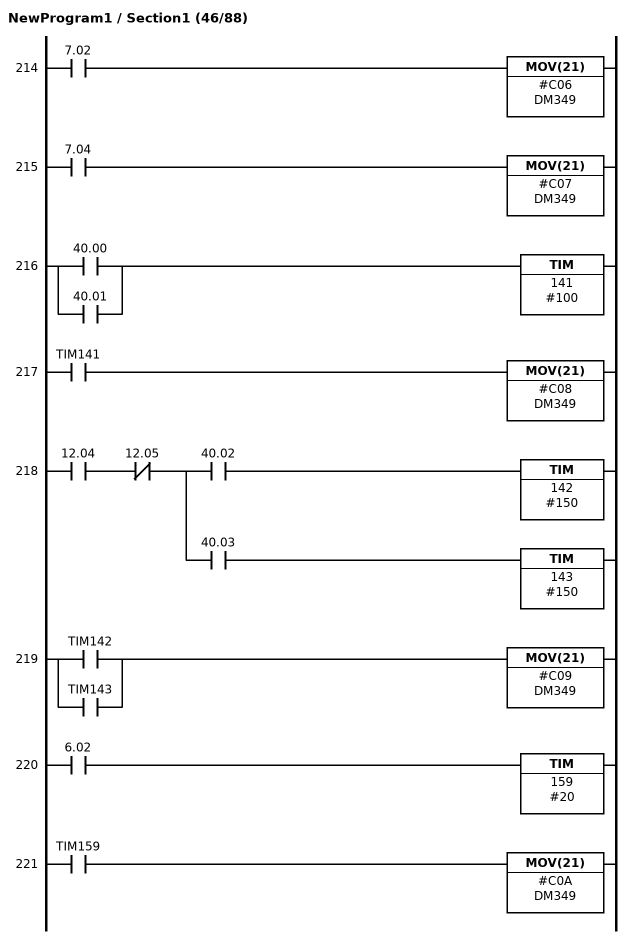
; rung 214
LD 7.02
MOV(21) #C06 DM349
; rung 215
LD 7.04
MOV(21) #C07 DM349
; rung 216
LD 40.00
OR 40.01
TIM 141 #100
; rung 217
LD TIM141
MOV(21) #C08 DM349
; rung 218
LD 12.04
ANDNOT 12.05
OUT TR0
AND 40.02
TIM 142 #150
LD TR0
AND 40.03
TIM 143 #150
; rung 219
LD TIM142
OR TIM143
MOV(21) #C09 DM349
; rung 220
LD 6.02
TIM 159 #20
; rung 221
LD TIM159
MOV(21) #C0A DM349

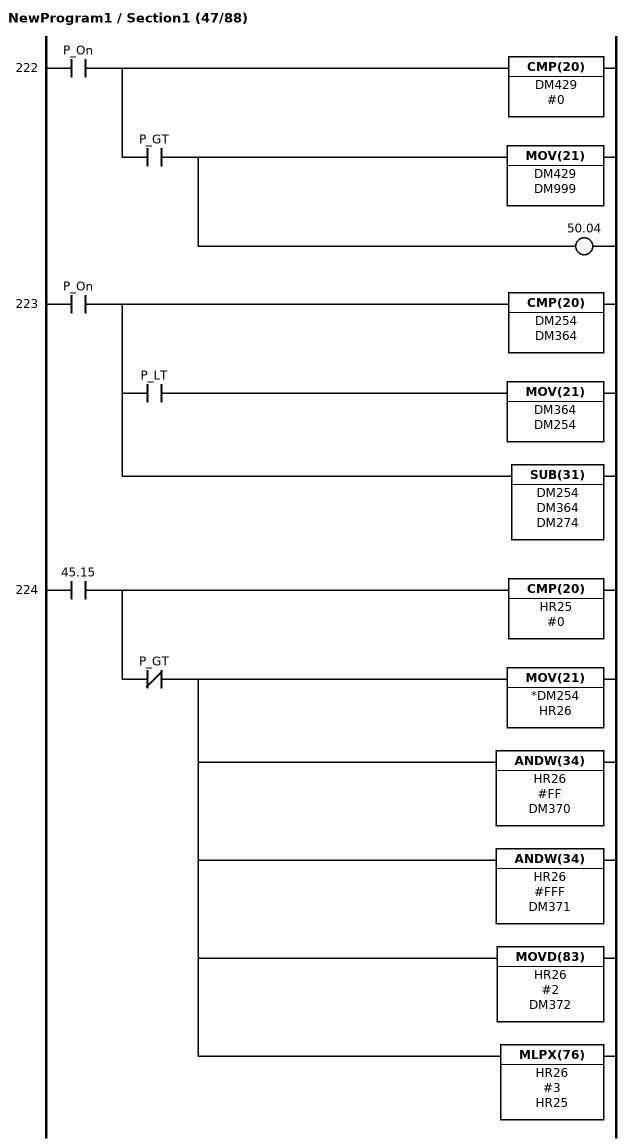
; rung 222
LD P_On
CMP(20) DM429 #0
AND P_GT
MOV(21) DM429 DM999
OUT 50.04
; rung 223
LD P_On
OUT TR0
CMP(20) DM254 DM364
AND P_LT
MOV(21) DM364 DM254
LD TR0
SUB(31) DM254 DM364 DM274
; rung 224
LD 45.15
CMP(20) HR25 #0
ANDNOT P_GT
MOV(21) *DM254 HR26
ANDW(34) HR26 #FF DM370
ANDW(34) HR26 #FFF DM371
MOVD(83) HR26 #2 DM372
MLPX(76) HR26 #3 HR25

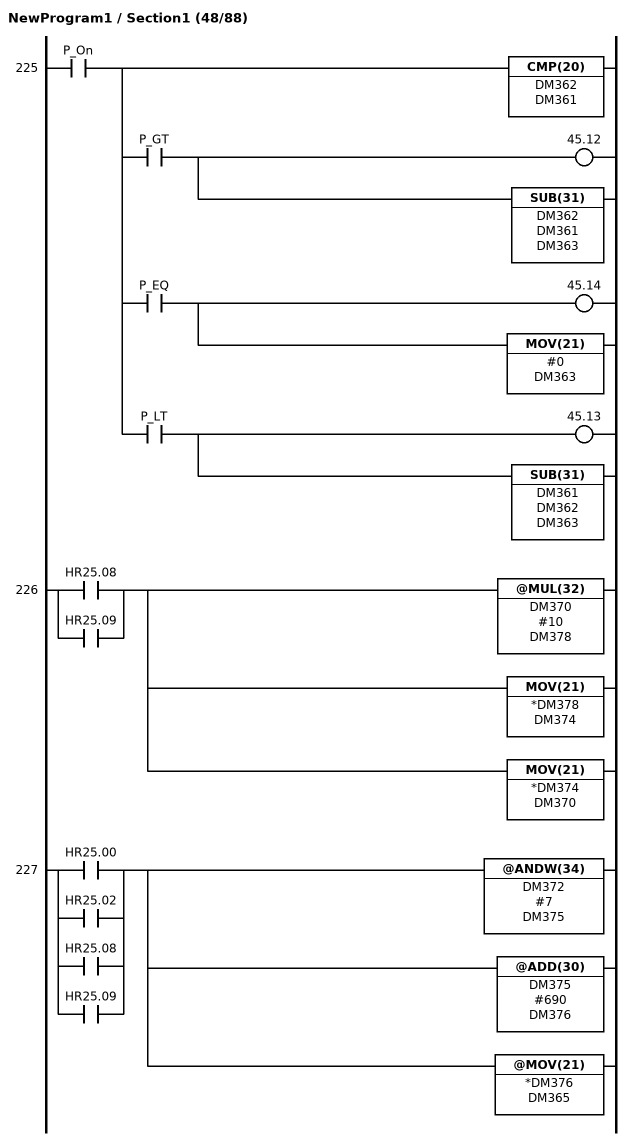
; rung 225
LD P_On
OUT TR0
CMP(20) DM362 DM361
AND P_GT
OUT 45.12
SUB(31) DM362 DM361 DM363
LD TR0
AND P_EQ
OUT 45.14
MOV(21) #0 DM363
LD TR0
AND P_LT
OUT 45.13
SUB(31) DM361 DM362 DM363
; rung 226
LD HR25.08
OR HR25.09
@MUL(32) DM370 #10 DM378
MOV(21) *DM378 DM374
MOV(21) *DM374 DM370
; rung 227
LD HR25.00
OR HR25.02
OR HR25.08
OR HR25.09
@ANDW(34) DM372 #7 DM375
@ADD(30) DM375 #690 DM376
@MOV(21) *DM376 DM365

